// TIA Portal V17 export
// export: Created 2025-01-08T13:55:32.0590774Z, ExportSetting WithDefaults, DisplayName Totally Integrated Automation Portal, DisplayVersion V17, DisplayName TIA Portal Openness, DisplayVersion V17, DisplayName TIA Portal Version Control Interface, DisplayVersion V17, DisplayName SINAMICS Startdrive Advanced, DisplayVersion V17 Update2, DisplayName SINAMICS Startdrive G130, G150, S120, S150, SINAMICS MV, S210, DisplayVersion V17 Update2, DisplayName SINAMICS Startdrive G110M, G120, G120C, G120D, G120P, G115D, DisplayVersion V17 Update2, DisplayName STEP 7 Professional, DisplayVersion V17, DisplayName STEP 7 Safety, DisplayVersion V17, DisplayName WinCC Advanced, DisplayVersion V17
FUNCTION_BLOCK "FB - Speed_Changer"   // FB37, LAD
{ S7_Optimized_Access := 'TRUE' }
VERSION : 0.1
// stored: AutoNumber true, IsIECCheckEnabled false, IsRetainMemResEnabled false, MemoryReserve 100, SetENOAutomatically false, UDAEnableTagReadback false
   VAR
      Speed_1_Pos : Bool;
      Speed_2_Pos : Bool;
      Speed_3_Pos : Bool;
      Speed_4_Pos : Bool;
      IEC_Timer_0_Instance { S7_SetPoint := 'True'} : TON_TIME;
      ResetSpeedEvents : Bool;
      Speed_5_Pos : Bool;
   END_VAR
   VAR_TEMP   // added for the SCL form of the ladder/FBD networks
      _w1 : Bool;
   END_VAR
BEGIN

REGION Network 1: Reset Speed Tags
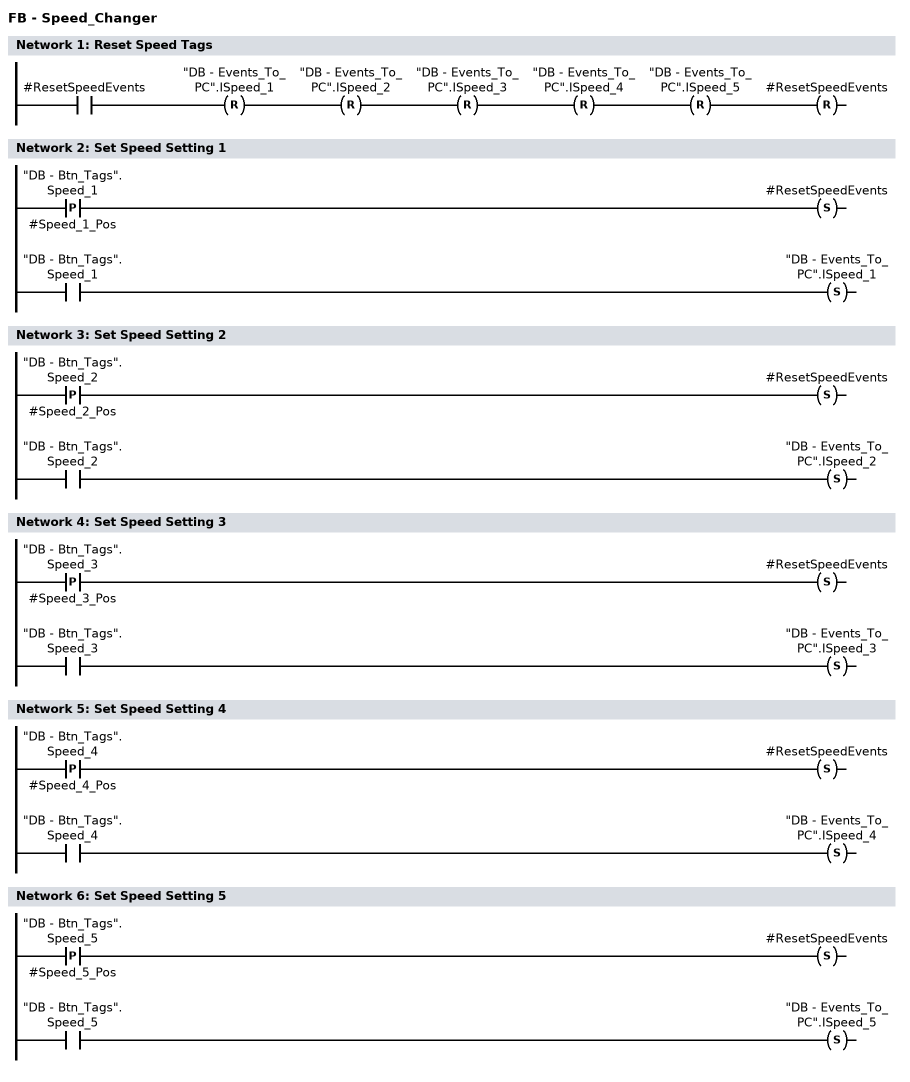
   RUNG wire#powerrail
      Contact( #ResetSpeedEvents )
      R_Coil( "DB - Events_To_PC".ISpeed_1 )
      R_Coil( "DB - Events_To_PC".ISpeed_2 )
      R_Coil( "DB - Events_To_PC".ISpeed_3 )
      R_Coil( "DB - Events_To_PC".ISpeed_4 )
      R_Coil( "DB - Events_To_PC".ISpeed_5 )
      R_Coil( #ResetSpeedEvents )
   END_RUNG
   // the same network as SCL:
   IF #ResetSpeedEvents THEN
       "DB - Events_To_PC".ISpeed_1 := FALSE;
       "DB - Events_To_PC".ISpeed_2 := FALSE;
       "DB - Events_To_PC".ISpeed_3 := FALSE;
       "DB - Events_To_PC".ISpeed_4 := FALSE;
       "DB - Events_To_PC".ISpeed_5 := FALSE;
       #ResetSpeedEvents := FALSE;
   END_IF;
END_REGION

REGION Network 2: Set Speed Setting 1
   RUNG wire#powerrail
      P_Contact(operand := "DB - Btn_Tags".Speed_1, bit := #Speed_1_Pos)
      S_Coil( #ResetSpeedEvents )
   END_RUNG
   RUNG wire#powerrail
      Contact( "DB - Btn_Tags".Speed_1 )
      S_Coil( "DB - Events_To_PC".ISpeed_1 )
   END_RUNG
   // the same network as SCL:
   #_w1 := "DB - Btn_Tags".Speed_1 AND NOT #Speed_1_Pos;   // rising edge of "DB - Btn_Tags".Speed_1
   #Speed_1_Pos := "DB - Btn_Tags".Speed_1;
   IF #_w1 THEN #ResetSpeedEvents := TRUE; END_IF;
   IF "DB - Btn_Tags".Speed_1 THEN "DB - Events_To_PC".ISpeed_1 := TRUE; END_IF;
END_REGION

REGION Network 3: Set Speed Setting 2
   RUNG wire#powerrail
      P_Contact(operand := "DB - Btn_Tags".Speed_2, bit := #Speed_2_Pos)
      S_Coil( #ResetSpeedEvents )
   END_RUNG
   RUNG wire#powerrail
      Contact( "DB - Btn_Tags".Speed_2 )
      S_Coil( "DB - Events_To_PC".ISpeed_2 )
   END_RUNG
   // the same network as SCL:
   #_w1 := "DB - Btn_Tags".Speed_2 AND NOT #Speed_2_Pos;   // rising edge of "DB - Btn_Tags".Speed_2
   #Speed_2_Pos := "DB - Btn_Tags".Speed_2;
   IF #_w1 THEN #ResetSpeedEvents := TRUE; END_IF;
   IF "DB - Btn_Tags".Speed_2 THEN "DB - Events_To_PC".ISpeed_2 := TRUE; END_IF;
END_REGION

REGION Network 4: Set Speed Setting 3
   RUNG wire#powerrail
      P_Contact(operand := "DB - Btn_Tags".Speed_3, bit := #Speed_3_Pos)
      S_Coil( #ResetSpeedEvents )
   END_RUNG
   RUNG wire#powerrail
      Contact( "DB - Btn_Tags".Speed_3 )
      S_Coil( "DB - Events_To_PC".ISpeed_3 )
   END_RUNG
   // the same network as SCL:
   #_w1 := "DB - Btn_Tags".Speed_3 AND NOT #Speed_3_Pos;   // rising edge of "DB - Btn_Tags".Speed_3
   #Speed_3_Pos := "DB - Btn_Tags".Speed_3;
   IF #_w1 THEN #ResetSpeedEvents := TRUE; END_IF;
   IF "DB - Btn_Tags".Speed_3 THEN "DB - Events_To_PC".ISpeed_3 := TRUE; END_IF;
END_REGION

REGION Network 5: Set Speed Setting 4
   RUNG wire#powerrail
      P_Contact(operand := "DB - Btn_Tags".Speed_4, bit := #Speed_4_Pos)
      S_Coil( #ResetSpeedEvents )
   END_RUNG
   RUNG wire#powerrail
      Contact( "DB - Btn_Tags".Speed_4 )
      S_Coil( "DB - Events_To_PC".ISpeed_4 )
   END_RUNG
   // the same network as SCL:
   #_w1 := "DB - Btn_Tags".Speed_4 AND NOT #Speed_4_Pos;   // rising edge of "DB - Btn_Tags".Speed_4
   #Speed_4_Pos := "DB - Btn_Tags".Speed_4;
   IF #_w1 THEN #ResetSpeedEvents := TRUE; END_IF;
   IF "DB - Btn_Tags".Speed_4 THEN "DB - Events_To_PC".ISpeed_4 := TRUE; END_IF;
END_REGION

REGION Network 6: Set Speed Setting 5
   RUNG wire#powerrail
      P_Contact(operand := "DB - Btn_Tags".Speed_5, bit := #Speed_5_Pos)
      S_Coil( #ResetSpeedEvents )
   END_RUNG
   RUNG wire#powerrail
      Contact( "DB - Btn_Tags".Speed_5 )
      S_Coil( "DB - Events_To_PC".ISpeed_5 )
   END_RUNG
   // the same network as SCL:
   #_w1 := "DB - Btn_Tags".Speed_5 AND NOT #Speed_5_Pos;   // rising edge of "DB - Btn_Tags".Speed_5
   #Speed_5_Pos := "DB - Btn_Tags".Speed_5;
   IF #_w1 THEN #ResetSpeedEvents := TRUE; END_IF;
   IF "DB - Btn_Tags".Speed_5 THEN "DB - Events_To_PC".ISpeed_5 := TRUE; END_IF;
END_REGION
END_FUNCTION_BLOCK
